{attribute 'qualified_only'}
{attribute 'strict'}
TYPE E_DiscreteValveFeedbackMode :
(
	noFeedback := 0,
	openedFeedback := 1,
	closedFeedback := 2,
	dualFeedback := 3
);
END_TYPE

(* stored: Version 1.1.0.1, ProductVersion 3.1.4024.10
   DUT E_DiscreteValveFeedbackMode: Id {ef082307-b571-4337-9420-de6f5004e905} *)
